PROGRAM MAIN
VAR
	BoolTestVar    : BOOL;
	ByteTestVar    : BYTE;
	USIntTestVar   : USINT;
	SIntTestVar    : SINT;
	UIntTestVar    : UINT;
	WordTestVar    : WORD;
	UDIntTestVar   : UDINT;
	ULIntTestVar   : ULINT;
	DWordTestVar   : DWORD;
	IntTestVar     : INT;
	DIntTestVar    : DINT;
	LIntTestVar    : LINT;
	RealTestVar    : REAL;
	LRealTestVar   : LREAL;
	StringTestVar  : STRING;
	WStringTestVar : WSTRING;
	TimeTestVar    : TIME;
	DTTestVar      : DT;
	TODTestVar     : TOD;
	
	RNG              : DRAND;
	UIntChangingVar  : UINT;
	LRealChangingVar : LREAL;
END_VAR

BoolTestVar := TRUE;

ByteTestVar := 9;

USIntTestVar := 12;

SIntTestVar := -21;

UIntTestVar := 32;

WordTestVar := 54;

UDIntTestVar := 44;

ULIntTestVar := 14;

DWordTestVar := 89;

IntTestVar := -23;

DIntTestVar := -23902;

LIntTestVar := -23903;

RealTestVar := 2.03032;

LRealTestVar := -4.202902239210;

StringTestVar := WSTRING_TO_STRING("String test var value");

WStringTestVar := "WString test var value with extra ümlauts";

TimeTestVar := T#14MS;

DTTestVar := DT#1972-03-29-00:00:00;

TODTestVar := TOD#15:36:30.123;

RNG();
LRealChangingVar := LRealChangingVar + RNG.Num;

RNG();
UIntChangingVar := UIntChangingVar + LREAL_TO_UINT(RNG.Num);

END_PROGRAM

(* stored: Version 1.1.0.1, ProductVersion 3.1.4024.6
   POU MAIN: Id {41b4b42b-7c31-49b3-abb2-c3d7dc97756e}, SpecialFunc None *)
